FUNCTION_BLOCK Room_State_Heating EXTENDS Room_State
VAR_INPUT
END_VAR
VAR_OUTPUT
END_VAR
VAR
END_VAR

METHOD OnInit
_ctx.io.out.bInletValve := FALSE;
_ctx.io.out.bOutletValve := FALSE;

_ctx.priv.bAbort := TRUE;
END_METHOD

END_FUNCTION_BLOCK

(* stored: Version 1.1.0.1
   POU Room_State_Heating: Id {c98dfd46-a1dc-427b-9523-1ac85e9186a3}, SpecialFunc None
   Method OnInit: Id {aa027ac0-d2d2-41a0-a2a1-be232fcb4334} *)
